FUNCTION_BLOCK SPLIT_MI_DO_S_Dual_SA (* Splits a DataPanel_MI_DO_S_Dual_SA into 2 DataPanel_MI_DO_S_Single_SA *)
  (* Standard: 61499-2; Description: Copyright (c) 2026 HR Agrartechnik GmbH SPDX-License-Identifier: EPL-2.0 *)
  (* Version 1.0, 2026-05-28, franz, HR Agrartechnik GmbH *)
  PACKAGE DataPanel::io::MI::DQ;
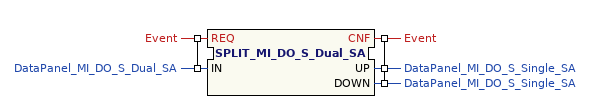
  EVENT_INPUT
    REQ WITH IN; (* Service Request *)
  END_EVENT
  EVENT_OUTPUT
    CNF WITH UP, DOWN; (* Confirmation of Requested Service *)
  END_EVENT
  VAR_INPUT
    IN : DataPanel::io::MI::DQ::DataPanel_MI_DO_S_Dual_SA; (* Dual Input *)
  END_VAR
  VAR_OUTPUT
    UP : DataPanel::io::MI::DQ::DataPanel_MI_DO_S_Single_SA; (* forward, up, right, clockwise *)
    DOWN : DataPanel::io::MI::DQ::DataPanel_MI_DO_S_Single_SA; (* backward, down, left, counter-clockwise *)
  END_VAR
  EC_STATES
    REQ : REQ -> CNF;
  END_STATES
  ALGORITHM REQ IN ST: (* Normally executed algorithm *)
UP.u8SAMember := IN.u8SAMember;
UP.Port := IN.Up;
DOWN.u8SAMember := IN.u8SAMember;
DOWN.Port := IN.Down;
  END_ALGORITHM
END_FUNCTION_BLOCK
